// TIA Portal V16 export
// export: Created 2022-02-28T20:45:46.3785498Z, ExportSetting WithDefaults, DisplayName Totally Integrated Automation Portal, DisplayVersion V16, DisplayName TIA Portal Version Control Interface, DisplayVersion V16, DisplayName TIA Portal Openness, DisplayVersion V16, DisplayName STEP 7 Professional, DisplayVersion V16, DisplayName STEP 7 Safety, DisplayVersion V16, DisplayName WinCC Advanced, DisplayVersion V16
DATA_BLOCK "06_Datos_Produccion"   // DB6
{ S7_Optimized_Access := 'TRUE' }
VERSION : 0.1
// stored: AutoNumber true, DBAccessibleFromOPCUA true, IsOnlyStoredInLoadMemory false, IsRetainMemResEnabled false, IsWriteProtectedInAS false, MemoryReserve 100
   VAR
      Datos_Prod_Pistilos : Struct
         Registro : "UDT_DatosProd";
         Pistilos_ONS : Array[1..10] of Bool;
      END_STRUCT;
      General : Struct
         Indice : Int;
      END_STRUCT;
   END_VAR
BEGIN
   Datos_Prod_Pistilos.Registro.Entradas.Longitud := 10;
END_DATA_BLOCK
